(*			
	RAFALOS
	Rafał Osajda		23.09.2025		TC 4024.66
	Struktura pomocnicza potrzeba do wiazania zmiennych
*)
TYPE ST_BaseComponent_HMI_Link :
STRUCT
	stBaseLoggerElement				: ST_BaseLoggerElement_HMI;
	stBaseComponent					: ST_BaseComponent_HMI;
END_STRUCT
END_TYPE

(* stored: Version 1.1.0.1
   DUT ST_BaseComponent_HMI_Link: Id {175661a4-aa2d-0650-1cf8-8a651fc90cc4} *)
